// TIA Portal project "plc2" (V17)
// Grundprojekt enthält nur die SPS

(* hardware
DEVICE "S71500/ET200MP-Station_1"  S7-1500 station
   slot 0: "Profilschiene_0"  Rack  6ES7 590-1***0-0AA0
   slot 0: "PM 190W 120/230VAC"  PM 190W 120/230VAC  6EP1333-4BA00
   slot 1: "PLC_2"  CPU 1516F-3 PN/DP  6ES7 516-3FN01-0AB0  V2.9
      slot 3: "CPU-Display_1"  6ES7591-1BA00-0AA0
      slot 32768: "PROFINET-Schnittstelle_1"  X1
      slot 33024: "PROFINET-Schnittstelle_2"  X2
      slot 34817: "Virtual CP interface port_1"  Virtual CP interface port  Virtual CP interface port
   slot 2: "DI 32x24VDC HF_1"  DI 32x24VDC HF  6ES7 521-1BL00-0AB0  V2.1
   slot 3: "DQ 32x24VDC/0.5A HF_1"  DQ 32x24VDC/0.5A HF  6ES7 522-1BL01-0AB0  V1.0
   slot 4: "AI 8xU/I/RTD/TC ST_1"  AI 8xU/I/RTD/TC ST  6ES7 531-7KF00-0AB0  V2.1
   slot 5: "AQ 4xU/I ST_1"  AQ 4xU/I ST  6ES7 532-5HD00-0AB0  V2.0
DEVICE "ET 200SP station_1"  ET 200SP-Station
   slot 0: "Rack_0"  Rack  6ES5 710-8MAx1
   slot 0: "IOdevice-1"  IM 155-6 PN/2 HF  6ES7 155-6AU01-0CN0  V4.2
   slot 1: "DI 8x24VDC HF_1"  DI 8x24VDC HF  6ES7 131-6BF00-0CA0  V2.0
      slot 1: "DI 8x24VDC HF_1"  DI 8x24VDC HF
   slot 2: "DI 8x24VDC HF_2"  DI 8x24VDC HF  6ES7 131-6BF00-0CA0  V2.0
      slot 1: "DI 8x24VDC HF_2"  DI 8x24VDC HF
   slot 3: "DQ 8x24VDC/0.5A HF_1"  DQ 8x24VDC/0.5A HF  6ES7 132-6BF00-0CA0  V2.0
      slot 1: "DQ 8x24VDC/0.5A HF_1"  DQ 8x24VDC/0.5A HF
   slot 4: "DQ 8x24VDC/0.5A HF_2"  DQ 8x24VDC/0.5A HF  6ES7 132-6BF00-0CA0  V2.0
      slot 1: "DQ 8x24VDC/0.5A HF_2"  DQ 8x24VDC/0.5A HF
   slot 5: "Server module_1"  Server module  6ES7 193-6PA00-0AA0  V1.1
      slot 1: "Server module_1"  Server module
   slot 127: "BA 2xRJ45"  BA 2xRJ45  6ES7 193-6AR00-0AA0  V0.0
      slot 1: "Port_1"  X1 P1 R  6ES7 193-6AR00-0AA0  V0.0
      slot 2: "Port_2"  X1 P2 R  6ES7 193-6AR00-0AA0  V0.0
DEVICE "SCALANCE XC-200"  SCALANCE X-Station
   slot 0: "SCALANCE X-Rack"  Rail
   slot 0: "Switch-1"  SCALANCE XC208  6GK5 208-0BA00-2AC2  V4.3
*)

// ===== PLC "PLC_2"  CPU 1516F-3 PN/DP =====

VAR_GLOBAL   // PLC tag table "Standard-Variablentabelle"
   "Clock_Byte" AT %MB0 : Byte;
   "Clock_10Hz" AT %M0.0 : Bool;
   "Clock_5Hz" AT %M0.1 : Bool;
   "Clock_2.5Hz" AT %M0.2 : Bool;
   "Clock_2Hz" AT %M0.3 : Bool;
   "Clock_1.25Hz" AT %M0.4 : Bool;
   "Clock_1Hz" AT %M0.5 : Bool;
   "Clock_0.625Hz" AT %M0.6 : Bool;
   "Clock_0.5Hz" AT %M0.7 : Bool;
   "tag1" AT %Q0.2 : Bool;
   "10S00" AT %I0.0 : Bool;
   "10S02" AT %I0.1 : Bool;
   "10H0_1" AT %Q0.0 : Bool;
   "10H0_2" AT %Q0.1 : Bool;
   "System_Byte" AT %MB1 : Byte;
   "FirstScan" AT %M1.0 : Bool;
   "DiagStatusUpdate" AT %M1.1 : Bool;
   "AlwaysTRUE" AT %M1.2 : Bool;
   "AlwaysFALSE" AT %M1.3 : Bool;
   "REQ_Toggle" AT %M4.0 : Bool;
   "Default_Speed" AT %MW6 : Int;
END_VAR

DATA_BLOCK "Data_to_PLC1"   // DB2
{ S7_Optimized_Access := 'FALSE' }
VERSION : 0.1
   VAR
      Motor_ON : Bool := true;
      Motor_Speed : Int := 500;
   END_VAR
BEGIN
END_DATA_BLOCK

DATA_BLOCK "PUT_Data_Block"   // DB3
{ S7_Optimized_Access := 'TRUE' }
VERSION : 0.1
// stored: InstanceOfName PUT_Communication
"PUT_Communication"
BEGIN
END_DATA_BLOCK

DATA_BLOCK "attack_input"   // DB4
{ S7_Optimized_Access := 'TRUE' }
VERSION : 0.1
   VAR
      Control_value_exceed : Bool;
      Control_value : Int := 2000;
      Rapid_value_change : Bool;
      "DOS attack" : Bool;
   END_VAR
BEGIN
END_DATA_BLOCK

DATA_BLOCK "Attacks_DB"   // DB5
{ S7_Optimized_Access := 'TRUE' }
VERSION : 0.1
// stored: InstanceOfName Attacks
"Attacks"
BEGIN
END_DATA_BLOCK

FUNCTION_BLOCK "PUT_Communication"   // FB1, LAD
{ S7_Optimized_Access := 'TRUE' }
VERSION : 0.1
BEGIN

REGION Network 1
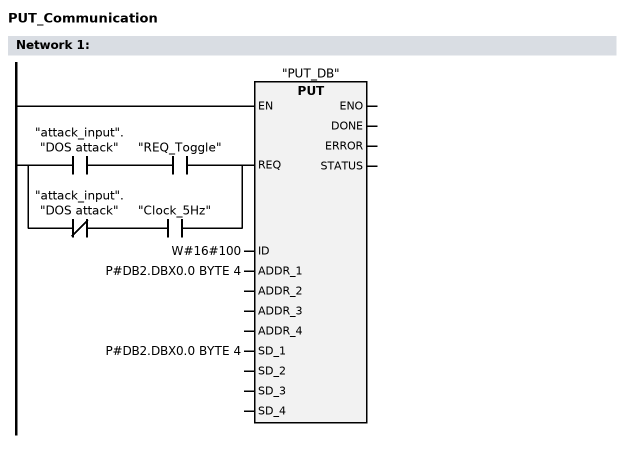
   "PUT_DB"(REQ := ("attack_input"."DOS attack" AND "REQ_Toggle") OR (NOT "attack_input"."DOS attack" AND "Clock_5Hz"),   // PUT
            ID := W#16#100,
            ADDR_1 := P#DB2.DBX0.0 BYTE 4,
            SD_1 := P#DB2.DBX0.0 BYTE 4);
END_REGION
END_FUNCTION_BLOCK

FUNCTION_BLOCK "Attacks"   // FB2, LAD
{ S7_Optimized_Access := 'TRUE' }
VERSION : 0.1
BEGIN

REGION Network 1: Attack 1: Control Value Exceed
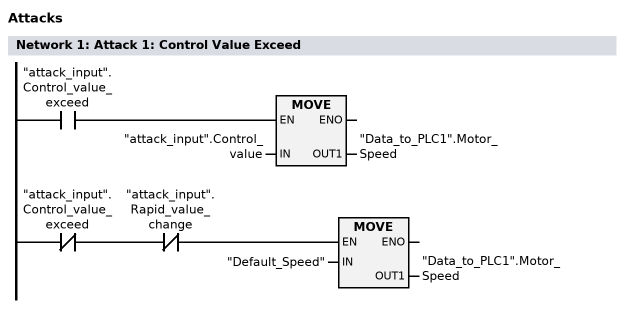
   RUNG wire#powerrail
      Contact( "attack_input".Control_value_exceed )
      Move(in := "attack_input".Control_value, out1 => "Data_to_PLC1".Motor_Speed)
   END_RUNG
   RUNG wire#powerrail
      I_Contact( "attack_input".Control_value_exceed )
      I_Contact( "attack_input".Rapid_value_change )
      Move(in := "Default_Speed", out1 => "Data_to_PLC1".Motor_Speed)
   END_RUNG
   // the same network as SCL:
   IF "attack_input".Control_value_exceed THEN
       "Data_to_PLC1".Motor_Speed := "attack_input".Control_value;
   END_IF;
   IF NOT "attack_input".Control_value_exceed AND NOT "attack_input".Rapid_value_change THEN
       "Data_to_PLC1".Motor_Speed := "Default_Speed";
   END_IF;
END_REGION

REGION Network 2 (SCL): ATTACK 2: Rapid Setpoint Changes
   IF "attack_input".Rapid_value_change THEN
       "Data_to_PLC1".Motor_Speed := "Data_to_PLC1".Motor_Speed + 100;
   END_IF;

   IF "Data_to_PLC1".Motor_Speed > 1400 AND "attack_input".Rapid_value_change THEN
       "Data_to_PLC1".Motor_Speed := 800;
   END_IF;
END_REGION
END_FUNCTION_BLOCK

ORGANIZATION_BLOCK "Main"   // OB1, FBD, ProgramCycle
TITLE = "Main Program Sweep (Cycle)"
{ S7_Optimized_Access := 'TRUE' }
VERSION : 0.1
   VAR_INPUT
      Initial_Call : Bool;   // Initial call of this OB
      Remanence : Bool;   // =True, if remanent data are available
   END_VAR
BEGIN

REGION Network 1
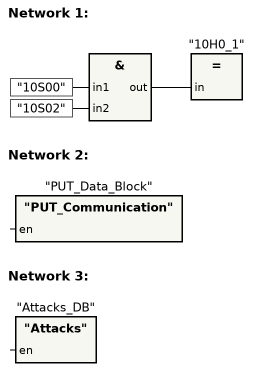
   "10H0_1" := "10S00" AND "10S02";
END_REGION

REGION Network 2
   "PUT_Data_Block"();   // "PUT_Communication"
END_REGION

REGION Network 3
   "Attacks_DB"();   // "Attacks"
END_REGION
END_ORGANIZATION_BLOCK